(* CODESYS project sensata_device_comm.library
   Company: Sensata Technologies
   Version: 0.0.1
   DocFormat: reStructuredText
   Placeholder: Sensata_Device_Comm
   Title: Sensata_Device_Comm

Project tree, tasks and I/O mapping:
  libraries: Sensata_Common, * (Sensata Technologies); Sensata_Utilities, * (Sensata Technologies); Tc2_Standard, * (Beckhoff Automation GmbH); Tc2_System, * (Beckhoff Automation GmbH); Tc2_Utilities, * (Beckhoff Automation GmbH); Tc3_Module, * (Beckhoff Automation GmbH)
  Abstract/
    function block FB_Device_Comm [ST]: M_init, M_LoadDevice, M_PowerDown, M_PowerUp, M_ReadDeviceOP, M_ReadSerialNumber, M_RunCommand, M_RunImpMethods, M_SetCurrentDevice
  Concrete/
    data type E_COHAP_Error
    function block FB_COHAP [ST]: M_init, M_LoadDevice, M_PowerDown, M_PowerUp, M_ReadDeviceOP, M_ReadSerialNumber, M_SetCurrentDevice, A_CommandRecovery, M_ParseValue, M_RouterHelper, M_RunCommand, M_RunImpMethods
  Interfaces/
    interface I_DeviceCommunicable: M_init, M_LoadDevice, M_PowerDown, M_PowerUp, M_ReadDeviceOP, M_ReadSerialNumber
  Project Information/
    function F_GetCompany [ST]
    function F_GetTitle [ST]
    function F_GetVersion [ST]
  Version/
    global variables Global_Version
  data type E_DataType
  data type ReturnParamKVP
  data type ST_CohapParam
  data type T_CohapParameterList
*)

// Concrete/E_COHAP_Error
{attribute 'qualified_only'}
{attribute 'strict'}
TYPE E_COHAP_Error :
(
	None := 0,
	
	CommandRouterError			:= 0100, // Error on the command router FB
	CommandFault 				:= 0101, // Command failed to execute
	
	FailedToLoadDevice 			:= 0200, // Unable Load new device information
	
	FailedToReadSerialNum		:=0300,// Read Serial num Fail
	FailedToReadDeviceOP		:=0301,// Read Device Op Fail
	FailedToPowerUp 			:= 0400, // Unable Load new device information
	FailedToPowerDown 			:= 0401, // Unable Load new device information
	
	FailedToRunImpMethods		:= 0500, //Unable to succesfully execute the runimpMethods function on DeviceComm CohapDevice.cs class
	FailedToExecuteRunCommand   := 0501  //Unable to execute the execute the RunCommand function on DeviceComm CohapDevice.cs class for the functionality we require
	
)UDINT;
END_TYPE

// E_DataType
TYPE E_DataType : (
    DT_INT,
    DT_REAL,
    DT_BOOL,
    DT_STRING,
    DT_DINT,
    DT_UDINT,
	DT_DATETIME,
	DT_DOUBLE,
	DT_INT64,
	DT_UINT,
	DT_ULINT //This is 64 bit equivalent
    // Add more as needed
);
END_TYPE

// ReturnParamKVP
TYPE ReturnParamKVP :
STRUCT
	VarName: STRING; // Key - Variable name
	DataType: E_DataType; // Value - Data type
END_STRUCT
END_TYPE

// ST_CohapParam
TYPE ST_CohapParam :
STRUCT
	strKey : T_MaxString;
	strValue : T_MaxString;//T_ApiParamValue;//T_MaxString;
END_STRUCT
END_TYPE

// T_CohapParameterList
TYPE T_CohapParameterList : ARRAY[0..9] OF ST_CohapParam; END_TYPE

// Version/Global_Version
{attribute 'TcGenerated'}
{attribute 'no-analysis'}
{attribute 'linkalways'}
// This function has been automatically generated from the project information.
VAR_GLOBAL CONSTANT
	{attribute 'const_non_replaced'}
	stLibVersion_Sensata_ASIC_Comm : ST_LibVersion := (iMajor := 0, iMinor := 0, iBuild := 1, iRevision := 0, nFlags := 0, sVersion := '0.0.1');
END_VAR

// Abstract/FB_Device_Comm
FUNCTION_BLOCK ABSTRACT FB_Device_Comm EXTENDS FB_Device IMPLEMENTS  I_DeviceCommunicable

VAR_INPUT
END_VAR
VAR_OUTPUT
END_VAR
VAR
END_VAR

{warning 'add method implementation '}
METHOD M_init : BOOL
VAR_INPUT
	(*channel*)
	udintChannel	: UDINT;
END_VAR
END_METHOD


METHOD M_LoadDevice : BOOL
VAR_INPUT
    strDevName: STRING ;//Device Name
END_VAR
END_METHOD


METHOD M_PowerDown : BOOL
VAR_INPUT
	str_devID: STRING;	
	Channel_Num:UDINT;
END_VAR
END_METHOD


METHOD M_PowerUp : BOOL
VAR_INPUT
	str_devID: STRING;	
	Channel_Num:UDINT;
	lrVsupply :LREAL;
	udintSalveadd: UDINT;

END_VAR
VAR_OUTPUT
	voltage: LREAL;	
	current:LREAL;
END_VAR
END_METHOD


METHOD M_ReadDeviceOP : BOOL
VAR_INPUT
	(* String representing Device ID *)
	str_deviceID: STRING;
	Channel_Num: UDINT;
END_VAR

VAR_OUTPUT
	(*  representing device op *)
	udint_MeasuredTemp: UDINT;
	udint_MeasuredPressure: UDINT;
END_VAR
M_ReadDeviceOP := TRUE;
THIS^.M_LogWarning('M_ReadDeviceOP not implemented!');
END_METHOD


METHOD M_ReadSerialNumber : BOOL
VAR_INPUT
	(* String representing Device ID *)
	str_deviceID: STRING;
	Channel_Num: UDINT;
END_VAR

VAR_OUTPUT
	(* udint representing read serial num from the device*)
	udintSerialNum: UDINT;
END_VAR
M_ReadSerialNumber := TRUE;
THIS^.M_LogWarning('M_ReadSerialNumber not implemented!');
END_METHOD

METHOD PUBLIC ABSTRACT M_RunCommand : BOOL
VAR_INPUT
	 strMethod :STRING;
	 aInputParam :T_CohapParameterList;//T_ApiParameterList//T_CohapParameterList
	 aExpectedOutputParamsList : ARRAY[0..9] OF ReturnParamKVP; // Adjust size as necessary;
END_VAR
VAR_OUTPUT
	 aoutputParam :T_CohapParameterList;//T_ApiParameterList//T_CohapParameterList
END_VAR
END_METHOD

METHOD PUBLIC ABSTRACT M_RunImpMethods : BOOL
VAR_INPUT
END_VAR
END_METHOD

METHOD PUBLIC ABSTRACT M_SetCurrentDevice : BOOL
VAR_INPUT
    strDevName: STRING ;//Device Name
END_VAR
END_METHOD

END_FUNCTION_BLOCK

// Interfaces/I_DeviceCommunicable
INTERFACE I_DeviceCommunicable

METHOD M_init : BOOL
VAR_INPUT
    udintChannel: UDINT ;//channel
END_VAR
END_METHOD

METHOD M_LoadDevice : BOOL
VAR_INPUT
    strDevName: STRING ;//Device Name
END_VAR
END_METHOD

METHOD M_PowerDown : BOOL
VAR_INPUT
	str_devID: STRING;	
	Channel_Num:UDINT;
END_VAR
END_METHOD

METHOD M_PowerUp : BOOL

VAR_INPUT
	str_devID: STRING;	
	Channel_Num:UDINT;
	lrVsupply :LREAL;
	udintSalveadd: UDINT;
	
END_VAR
VAR_OUTPUT
	voltage: LREAL;	
	current:LREAL;
END_VAR
END_METHOD

METHOD M_ReadDeviceOP : BOOL
VAR_INPUT
	(* String representing Device ID *)
	str_deviceID: STRING;
	Channel_Num: UDINT;
END_VAR

VAR_OUTPUT
	(*  representing device op *)
	udint_MeasuredTemp: UDINT;
	udint_MeasuredPressure: UDINT;
END_VAR
END_METHOD

METHOD M_ReadSerialNumber : BOOL
VAR_INPUT
	(* String representing Device ID *)
	str_deviceID: STRING;
	Channel_Num: UDINT;
END_VAR

VAR_OUTPUT
	(* udint representing read serial num from the device*)
	udintSerialNum: UDINT;
END_VAR
END_METHOD

END_INTERFACE

// Concrete/FB_COHAP
FUNCTION_BLOCK FB_COHAP EXTENDS FB_Device_Comm IMPLEMENTS  I_DeviceCommunicable

VAR_INPUT
	(* Reference to an FB_CommandRouter function block to send commands
		to a command router in the API. *)
	fbApi : REFERENCE TO FB_CommandRouter;
END_VAR
VAR_OUTPUT
END_VAR
VAR
	
// Connectable
	bApiConnected: BOOL; (* TRUE if the API is connected. *)
	bConnected: BOOL; (* TRUE if the hipot is connected. *)
	bConnecting: BOOL; (* TRUE while the connect command is running. *)
	bDisconnecting: BOOL; (* TRUE while the disconnect command is running. *)
	
	enumProgramState: E_PROGRAMSTATE; // Value of P_enumProgramState
	bRouterBusy: BOOL; // TRUE while M_RouterHelper is being used by a method
	bResetBusy: BOOL; // Value of P_bResetBusy
	
	
	intInitStep: INT;
	intLoadDeviceStep: INT;
	intPowerUpStep: INT;
	intPowerDownStep: INT;
	intReadDeviceOPStep: INT;
	intReadDeviceSNStep: INT;
	intRouterHelperStep: INT;
	intMSetCurrentDeviceStep : INT;
	intMRunCommandStep : INT;
	intMRunImpMethodsStep : INT;
	
	
	bLoadDeviceBusy: BOOL;
	bInitBusy: BOOL;
	bPowerUpBusy: BOOL;
	bPowerDownBusy: BOOL;
	bReadDeviceOPBusy:BOOL;
	bReadDeviceSerialNumberBusy:BOOL;
	bRouterHelperBusy: BOOL;
	bSetCurrentDeviceBusy : BOOL;
	bMRunCommandBusy : BOOL;
	bRunImpMethodsBusy : BOOL;
	
END_VAR


A_CommandRecovery();

METHOD M_init : BOOL
VAR_INPUT
    udintChannel: UDINT ;//channel
END_VAR

VAR CONSTANT
	_strCOMMAND_NAME : T_MaxString	:= 'init'; // Name of the API method
	_timeCOMMAND_TIMEOUT : TIME		:= T#5S; // Max time to receive API response
	_strSTART_MSG : T_MaxString		:= 'initializing DUT '; // Prints when method starts
	_strEND_MSG : T_MaxString		:= 'DUT structure initialized'; // Prints when method finishes
	_udintERROR_ID : UDINT			:= E_COHAP_Error.FailedToLoadDevice; // Error ID to set if command fails
	_strERROR_MSG : T_MaxString		:= 'Failed to initialize!'; // Error message to set if command fails
END_VAR
VAR_INST
	_inst_arrParams: T_ApiParameterList; // Parameters array
	_inst_arrOutputs: T_ApiParameterList; // Outputs array
	_inst_strRet: T_ApiParamValue; // Return string from the router
	_inst_intStep: INT; // Current method step
	_inst_fbParams: FB_ApiParamBuilder; // Parameter builder FB
END_VAR
VAR
	_bComplete: BOOL; // True if the routing finishes
	_intRet: INT; // Return string converted to an integer
	_bResult : BOOL; // Output of the method
END_VAR
_inst_intStep:=intInitStep;
bInitBusy:=TRUE;

_bResult:=FALSE;
CASE _inst_intStep OF
	0: // Wait for no error and router not busy
		IF NOT THIS^.P_bError AND NOT bRouterBusy THEN
			bRouterBusy := TRUE;
			_inst_intStep := _inst_intStep + 10;
		END_IF
		
	10: // Initialize parameters
		THIS^.M_LogMessage(_strSTART_MSG);
		_inst_fbParams.M_ClearParameters();
		// ADD ANY PARAMETERS HERE
		_inst_fbParams.M_AddParameter('channel', udintChannel);
		
		_inst_fbParams.M_OutputToParameterList(_inst_arrParams);
		_inst_intStep := _inst_intStep + 10;
		
	20: // Route the command
		_bComplete := M_RouterHelper(
			_in_strMethodName := _strCOMMAND_NAME, 
			_in_timeTimeout := _timeCOMMAND_TIMEOUT,
			_inout_arrParams := _inst_arrParams,
			_inout_arrOutputs := _inst_arrOutputs,
			_out_strReturnValue=>_inst_strRet);
		
		// If route completed, move to next step
		IF _bComplete THEN
			_inst_intStep := _inst_intStep + 10;
			bRouterBusy := FALSE;
		ELSIF THIS^.P_bError THEN
			_inst_intStep := 0;
			bRouterBusy := FALSE;
		END_IF
		
	30: // Parse results
		_intRet := STRING_TO_INT(_inst_strRet);
		IF _intRet > 0 THEN
			_bResult := TRUE;
			THIS^.M_LogMessage(_strEND_MSG);
			// DO ANY PARSING HERE
			_inst_fbParams.M_LoadFromParameterList(_inst_arrOutputs);
		
		// Set error if command failed
	
		ELSE
			THIS^.M_SetError(_udintERROR_ID, _strERROR_MSG);
		END_IF
		
		// Go back to start
		_inst_intStep := 0;
END_CASE
M_init := _bResult;
intInitStep:=_inst_intStep;
END_METHOD

METHOD M_LoadDevice : BOOL
VAR_INPUT
    strDevName: STRING ;//Device Name
END_VAR

VAR CONSTANT
	_strCOMMAND_NAME : T_MaxString	:= 'LoadDevice'; // Name of the API method
	_timeCOMMAND_TIMEOUT : TIME		:= T#5S; // Max time to receive API response
	_strSTART_MSG : T_MaxString		:= 'Load a new device to test'; // Prints when method starts
	_strEND_MSG : T_MaxString		:= 'Device details loaded'; // Prints when method finishes
	_udintERROR_ID : UDINT			:= E_COHAP_Error.FailedToLoadDevice; // Error ID to set if command fails
	_strERROR_MSG : T_MaxString		:= 'Failed to connect!'; // Error message to set if command fails
END_VAR
VAR_INST
	_inst_arrParams: T_ApiParameterList; // Parameters array
	_inst_arrOutputs: T_ApiParameterList; // Outputs array
	_inst_strRet: T_ApiParamValue; // Return string from the router
	_inst_intStep: INT; // Current method step
	_inst_fbParams: FB_ApiParamBuilder; // Parameter builder FB
END_VAR
VAR
	_bComplete: BOOL; // True if the routing finishes
	_intRet: INT; // Return string converted to an integer
	_bResult : BOOL; // Output of the method
END_VAR
_inst_intStep:=intLoadDeviceStep;
bLoadDeviceBusy:=TRUE;

_bResult := FALSE;
CASE _inst_intStep OF
	0: // Wait for no error and router not busy
		IF NOT THIS^.P_bError AND NOT bRouterBusy THEN
			bRouterBusy := TRUE;
			_inst_intStep := _inst_intStep + 10;
		END_IF
		
	10: // Initialize parameters
		THIS^.M_LogMessage(_strSTART_MSG);
		_inst_fbParams.M_ClearParameters();
		// ADD ANY PARAMETERS HERE
		_inst_fbParams.M_AddParameter('devID', strDevName);
		
		_inst_fbParams.M_OutputToParameterList(_inst_arrParams);
		_inst_intStep := _inst_intStep + 10;
		
	20: // Route the command
		_bComplete := M_RouterHelper(
			_in_strMethodName := _strCOMMAND_NAME, 
			_in_timeTimeout := _timeCOMMAND_TIMEOUT,
			_inout_arrParams := _inst_arrParams,
			_inout_arrOutputs := _inst_arrOutputs,
			_out_strReturnValue=>_inst_strRet);
		
		// If route completed, move to next step
		IF _bComplete THEN
			_inst_intStep := _inst_intStep + 10;
			bRouterBusy := FALSE;
		ELSIF THIS^.P_bError THEN
			_inst_intStep := 0;
			bRouterBusy := FALSE;
		END_IF
		
	30: // Parse results
		_intRet := STRING_TO_INT(_inst_strRet);
		IF _intRet > 0 THEN
			_bResult := TRUE;
			THIS^.M_LogMessage(_strEND_MSG);
			// DO ANY PARSING HERE
			_inst_fbParams.M_LoadFromParameterList(_inst_arrOutputs);
		
		// Set error if command failed
	
		ELSE
			THIS^.M_SetError(_udintERROR_ID, _strERROR_MSG);
		END_IF
		
		// Go back to start
		_inst_intStep := 0;
END_CASE
M_LoadDevice := _bResult;
intLoadDeviceStep:=_inst_intStep;
END_METHOD


METHOD M_PowerDown : BOOL
VAR_INPUT
	str_devID: STRING;	
	Channel_Num:UDINT;

END_VAR
VAR CONSTANT
	_strCOMMAND_NAME : T_MaxString	:= 'Powerdown'; // Name of the API method
	_timeCOMMAND_TIMEOUT : TIME		:= T#5S; // Max time to receive API response
	_strSTART_MSG : T_MaxString		:= 'Powering Down device'; // Prints when method starts
	_strEND_MSG : T_MaxString		:= 'Device Powered Down'; // Prints when method finishes
	_udintERROR_ID : UDINT			:= E_COHAP_Error.FailedToPowerDown; // Error ID to set if command fails
	_strERROR_MSG : T_MaxString		:= 'Failed to Power Down!'; // Error message to set if command fails
END_VAR
VAR_INST
	_inst_arrParams: T_ApiParameterList; // Parameters array
	_inst_arrOutputs: T_ApiParameterList; // Outputs array
	_inst_strRet: T_ApiParamValue; // Return string from the router
	_inst_intStep: INT; // Current method step
	_inst_fbParams: FB_ApiParamBuilder; // Parameter builder FB
END_VAR
VAR
	_bComplete: BOOL; // True if the routing finishes
	_intRet: INT; // Return string converted to an integer
	_bResult : BOOL; // Output of the method
END_VAR
_inst_intStep := intPowerDownStep;
bPowerDownBusy := TRUE;

_bResult := FALSE;
CASE _inst_intStep OF
	0: // Wait for no error and router not busy
		IF NOT THIS^.P_bError AND NOT bRouterBusy THEN
			bRouterBusy := TRUE;
			_inst_intStep := _inst_intStep + 10;
		END_IF
		
	10: // Initialize parameters
		THIS^.M_LogMessage(_strSTART_MSG);
		_inst_fbParams.M_ClearParameters();
		// ADD ANY PARAMETERS HERE
		
		_inst_fbParams.M_AddParameter('devID', str_devID);
		_inst_fbParams.M_AddParameter('channel', Channel_Num);
		_inst_fbParams.M_OutputToParameterList(_inst_arrParams);
		_inst_intStep := _inst_intStep + 10;
		
	20: // Route the command
		_bComplete := M_RouterHelper(
			_in_strMethodName := _strCOMMAND_NAME, 
			_in_timeTimeout := _timeCOMMAND_TIMEOUT,
			_inout_arrParams := _inst_arrParams,
			_inout_arrOutputs := _inst_arrOutputs,
			_out_strReturnValue=>_inst_strRet);
		
		// If route completed, move to next step
		IF _bComplete THEN
			_inst_intStep := _inst_intStep + 10;
			bRouterBusy := FALSE;
		ELSIF THIS^.P_bError THEN
			_inst_intStep := 0;
			bRouterBusy := FALSE;
		END_IF
		
	30: // Parse results
		_intRet := STRING_TO_INT(_inst_strRet);
		IF _intRet > 0 THEN
			_bResult := TRUE;
			THIS^.M_LogMessage(_strEND_MSG);
			// DO ANY PARSING HERE
			_inst_fbParams.M_LoadFromParameterList(_inst_arrOutputs);
		
		// Set error if command failed
	
		ELSE
			THIS^.M_SetError(_udintERROR_ID, _strERROR_MSG);
		END_IF
		
		// Go back to start
		_inst_intStep := 0;
END_CASE
M_PowerDown := _bResult;
intPowerDownStep:=_inst_intStep;
END_METHOD

METHOD M_PowerUp : BOOL
VAR_INPUT
	str_devID: STRING;	
	Channel_Num:UDINT;
	lrVsupply :LREAL;
	udintSalveadd: UDINT;
END_VAR
VAR_OUTPUT
	voltage: LREAL;	
	current:LREAL;
END_VAR
VAR CONSTANT
	_strCOMMAND_NAME : T_MaxString	:= 'Powerup'; // Name of the API method
	_timeCOMMAND_TIMEOUT : TIME		:= T#5S; // Max time to receive API response
	_strSTART_MSG : T_MaxString		:= 'Powering Up device'; // Prints when method starts
	_strEND_MSG : T_MaxString		:= 'Device Powered Up'; // Prints when method finishes
	_udintERROR_ID : UDINT			:= E_COHAP_Error.FailedToPowerUp; // Error ID to set if command fails
	_strERROR_MSG : T_MaxString		:= 'Failed to Power Up!'; // Error message to set if command fails
END_VAR
VAR_INST
	_inst_arrParams: T_ApiParameterList; // Parameters array
	_inst_arrOutputs: T_ApiParameterList; // Outputs array
	_inst_strRet: T_ApiParamValue; // Return string from the router
	_inst_intStep: INT; // Current method step
	_inst_fbParams: FB_ApiParamBuilder; // Parameter builder FB
END_VAR
VAR
	_bComplete: BOOL; // True if the routing finishes
	_intRet: INT; // Return string converted to an integer
	_bResult : BOOL; // Output of the method
END_VAR
_inst_intStep := intPowerUpStep;
bPowerUpBusy := TRUE;

_bResult := FALSE;
CASE _inst_intStep OF
	0: // Wait for no error and router not busy
		IF NOT THIS^.P_bError AND NOT bRouterBusy THEN
			bRouterBusy := TRUE;
			_inst_intStep := _inst_intStep + 10;
		END_IF
		
	10: // Initialize parameters
		THIS^.M_LogMessage(_strSTART_MSG);
		_inst_fbParams.M_ClearParameters();
		// ADD ANY PARAMETERS HERE
		
		_inst_fbParams.M_AddParameter('devID', str_devID);
		_inst_fbParams.M_AddParameter('channel', Channel_Num);
		_inst_fbParams.M_AddParameter('VSupply', lrVsupply);
		_inst_fbParams.M_AddParameter('slaveadd', udintSalveadd);
		_inst_fbParams.M_OutputToParameterList(_inst_arrParams);
		_inst_intStep := _inst_intStep + 10;
		
	20: // Route the command
		_bComplete := M_RouterHelper(
			_in_strMethodName := _strCOMMAND_NAME, 
			_in_timeTimeout := _timeCOMMAND_TIMEOUT,
			_inout_arrParams := _inst_arrParams,
			_inout_arrOutputs := _inst_arrOutputs,
			_out_strReturnValue=>_inst_strRet);
		
		// If route completed, move to next step
		IF _bComplete THEN
			_inst_intStep := _inst_intStep + 10;
			bRouterBusy := FALSE;
		ELSIF THIS^.P_bError THEN
			_inst_intStep := 0;
			bRouterBusy := FALSE;
		END_IF
		
	30: // Parse results
		_intRet := STRING_TO_INT(_inst_strRet);
		IF _intRet > 0 THEN
			_bResult := TRUE;
			THIS^.M_LogMessage(_strEND_MSG);
			// DO ANY PARSING HERE
			_inst_fbParams.M_LoadFromParameterList(_inst_arrOutputs);
			voltage := _inst_fbParams.M_ParseDouble(_inst_fbParams.M_GetParameter('Respvoltage'));
			current := _inst_fbParams.M_ParseDouble(_inst_fbParams.M_GetParameter('Respcurrent'));
		// Set error if command failed
	
		ELSE
			THIS^.M_SetError(_udintERROR_ID, _strERROR_MSG);
		END_IF
		
		// Go back to start
		_inst_intStep := 0;
END_CASE
M_PowerUp := _bResult;
intPowerUpStep:=_inst_intStep;
END_METHOD


(* This method takes deviceID as input as passes it to the COHAP API library to get the Device OP *)
METHOD M_ReadDeviceOP : BOOL
VAR_INPUT
	(* String representing Device ID *)
	str_deviceID: STRING;
	Channel_Num: UDINT;
END_VAR

VAR_OUTPUT
	(*  representing device op *)
	udint_MeasuredTemp: UDINT;
	udint_MeasuredPressure: UDINT;
END_VAR
VAR CONSTANT
	_strCOMMAND_NAME : T_MaxString	:= 'ReadDeviceOutput'; // Name of the API method
	_timeCOMMAND_TIMEOUT : TIME		:= T#7S; // Max time to receive API response
	_strSTART_MSG : T_MaxString		:= 'Reading Device output'; // Prints when method starts
	_strEND_MSG : T_MaxString		:= 'Completed device OP read'; // Prints when method finishes
	_udintERROR_ID : UDINT			:= E_COHAP_Error.FailedToReadDeviceOP; // Error ID to set if command fails
	_strERROR_MSG : T_MaxString		:= 'Failed to read Device output!'; // Error message to set if command fails
END_VAR
VAR_INST
	_inst_arrParams: T_ApiParameterList; // Parameters array
	_inst_arrOutputs: T_ApiParameterList; // Outputs array
	_inst_strRet: T_ApiParamValue; // Return string from the router
	_inst_intStep: INT; // Current method step
	_inst_fbParams: FB_ApiParamBuilder; // Parameter builder FB
END_VAR
VAR
	_bComplete: BOOL; // True if the routing finishes
	_intRet: INT; // Return string converted to an integer
	_bResult : BOOL; // Output of the method
END_VAR
_inst_intStep := intReadDeviceOPStep;
bReadDeviceOPBusy := TRUE;

_bResult := FALSE;
CASE _inst_intStep OF
	0: // Wait for no error and router not busy
		IF NOT THIS^.P_bError AND NOT bRouterBusy THEN
			bRouterBusy := TRUE;
			_inst_intStep := _inst_intStep + 10;
		END_IF
		
	10: // Initialize parameters
		THIS^.M_LogMessage(_strSTART_MSG);
		_inst_fbParams.M_ClearParameters();
		// ADD ANY PARAMETERS HERE
		_inst_fbParams.M_AddParameter('DeviceID', str_deviceID);
		_inst_fbParams.M_AddParameter('channel', Channel_Num);
		_inst_fbParams.M_OutputToParameterList(_inst_arrParams);
		_inst_intStep := _inst_intStep + 10;
		
	20: // Route the command
		_bComplete := M_RouterHelper(
			_in_strMethodName := _strCOMMAND_NAME, 
			_in_timeTimeout := _timeCOMMAND_TIMEOUT,
			_inout_arrParams := _inst_arrParams,
			_inout_arrOutputs := _inst_arrOutputs,
			_out_strReturnValue=>_inst_strRet);
		
		// If route completed, move to next step
		IF _bComplete THEN
			_inst_intStep := _inst_intStep + 10;
			bRouterBusy := FALSE;
		ELSIF THIS^.P_bError THEN
			_inst_intStep := 0;
			bRouterBusy := FALSE;
		END_IF
		
	30: // Parse results
		_intRet := STRING_TO_INT(_inst_strRet);
		IF _intRet > 0 THEN
			_bResult := TRUE;
			THIS^.M_LogMessage(_strEND_MSG);
			// DO ANY PARSING HERE
			_inst_fbParams.M_LoadFromParameterList(_inst_arrOutputs);
			udint_MeasuredTemp := _inst_fbParams.M_ParseUint(_inst_fbParams.M_GetParameter('OutputTemp'));
			udint_MeasuredPressure := _inst_fbParams.M_ParseUint(_inst_fbParams.M_GetParameter('OutputPress'));		
		// Set error if command failed
	
		ELSE
			THIS^.M_SetError(_udintERROR_ID, _strERROR_MSG);
		END_IF
		
		// Go back to start
		_inst_intStep := 0;
END_CASE
M_ReadDeviceOP := _bResult;
intReadDeviceOPStep:=_inst_intStep;
END_METHOD




(* This method takes deviceID as input as passes it to the COHAP API library to get the serial number *)
METHOD M_ReadSerialNumber : BOOL
VAR_INPUT
	(* String representing Device ID *)
	str_deviceID: STRING;
	Channel_Num: UDINT;

END_VAR

VAR_OUTPUT
	(* udint representing read serial num from the device*)
	udintSerialNum: UDINT;
END_VAR
VAR CONSTANT
	_strCOMMAND_NAME : T_MaxString	:= 'ReadSerialNumber'; // Name of the API method
	_timeCOMMAND_TIMEOUT : TIME		:= T#7S; // Max time to receive API response
	_strSTART_MSG : T_MaxString		:= 'Reading Device Serialnumber'; // Prints when method starts
	_strEND_MSG : T_MaxString		:= 'Completed Serial Num read'; // Prints when method finishes
	_udintERROR_ID : UDINT			:= E_COHAP_Error.FailedToReadSerialNum; // Error ID to set if command fails
	_strERROR_MSG : T_MaxString		:= 'Failed to read serial number!'; // Error message to set if command fails
END_VAR
VAR_INST
	_inst_arrParams: T_ApiParameterList; // Parameters array
	_inst_arrOutputs: T_ApiParameterList; // Outputs array
	_inst_strRet: T_ApiParamValue; // Return string from the router
	_inst_intStep: INT; // Current method step
	_inst_fbParams: FB_ApiParamBuilder; // Parameter builder FB
END_VAR
VAR
	_bComplete: BOOL; // True if the routing finishes
	_intRet: INT; // Return string converted to an integer
	_bResult : BOOL; // Output of the method
END_VAR
_inst_intStep := intReadDeviceSNStep;
bReadDeviceSerialNumberBusy := TRUE;

_bResult := FALSE;
CASE _inst_intStep OF
	0: // Wait for no error and router not busy
		IF NOT THIS^.P_bError AND NOT bRouterBusy THEN
			bRouterBusy := TRUE;
			_inst_intStep := _inst_intStep + 10;
		END_IF
		
	10: // Initialize parameters
		THIS^.M_LogMessage(_strSTART_MSG);
		_inst_fbParams.M_ClearParameters();
		// ADD ANY PARAMETERS HERE
		_inst_fbParams.M_AddParameter('DeviceID', str_deviceID);
		_inst_fbParams.M_AddParameter('channel', Channel_Num);
		_inst_fbParams.M_OutputToParameterList(_inst_arrParams);
		_inst_intStep := _inst_intStep + 10;
		
	20: // Route the command
		_bComplete := M_RouterHelper(
			_in_strMethodName := _strCOMMAND_NAME, 
			_in_timeTimeout := _timeCOMMAND_TIMEOUT,
			_inout_arrParams := _inst_arrParams,
			_inout_arrOutputs := _inst_arrOutputs,
			_out_strReturnValue=>_inst_strRet);
		
		// If route completed, move to next step
		IF _bComplete THEN
			_inst_intStep := _inst_intStep + 10;
			bRouterBusy := FALSE;
		ELSIF THIS^.P_bError THEN
			_inst_intStep := 0;
			bRouterBusy := FALSE;
		END_IF
		
	30: // Parse results
		_intRet := STRING_TO_INT(_inst_strRet);
		IF _intRet > 0 THEN
			_bResult := TRUE;
			THIS^.M_LogMessage(_strEND_MSG);
			// DO ANY PARSING HERE
			_inst_fbParams.M_LoadFromParameterList(_inst_arrOutputs);
			udintSerialNum := _inst_fbParams.M_ParseUint(_inst_fbParams.M_GetParameter('serialNumber'));
					
		// Set error if command failed
	
		ELSE
			THIS^.M_SetError(_udintERROR_ID, _strERROR_MSG);
		END_IF
		
		// Go back to start
		_inst_intStep := 0;
END_CASE
M_ReadSerialNumber := _bResult;
intReadDeviceSNStep:=_inst_intStep;
END_METHOD

METHOD M_SetCurrentDevice : BOOL
VAR_INPUT
    strDevName: STRING ;//Device Name
END_VAR

VAR CONSTANT
	_strCOMMAND_NAME : T_MaxString	:= 'SetCurrentDevice'; // Name of the API method
	_timeCOMMAND_TIMEOUT : TIME		:= T#30S; // Max time to receive API response
	_strSTART_MSG : T_MaxString		:= 'Load a new device to test'; // Prints when method starts
	_strEND_MSG : T_MaxString		:= 'Device details loaded'; // Prints when method finishes
	_udintERROR_ID : UDINT			:= E_COHAP_Error.FailedToLoadDevice; // Error ID to set if command fails
	_strERROR_MSG : T_MaxString		:= 'Failed to connect!'; // Error message to set if command fails
END_VAR
VAR_INST
	_inst_arrParams: T_ApiParameterList; // Parameters array
	_inst_arrOutputs: T_ApiParameterList; // Outputs array
	_inst_strRet: T_ApiParamValue; // Return string from the router
	_inst_intStep: INT; // Current method step
	_inst_fbParams: FB_ApiParamBuilder; // Parameter builder FB
END_VAR
VAR
	_bComplete: BOOL; // True if the routing finishes
	_intRet: INT; // Return string converted to an integer
	_bResult : BOOL; // Output of the method
END_VAR
_inst_intStep := intMSetCurrentDeviceStep;
bSetCurrentDeviceBusy := TRUE;

_bResult := FALSE;
CASE _inst_intStep OF
	0: // Wait for no error and router not busy
		IF NOT THIS^.P_bError AND NOT bRouterBusy THEN
			bRouterBusy := TRUE;
			_inst_intStep := _inst_intStep + 10;
		END_IF
		
	10: // Initialize parameters
		THIS^.M_LogMessage(_strSTART_MSG);
		_inst_fbParams.M_ClearParameters();
		// ADD ANY PARAMETERS HERE
		_inst_fbParams.M_AddParameter('DeviceName', strDevName);
		
		_inst_fbParams.M_OutputToParameterList(_inst_arrParams);
		_inst_intStep := _inst_intStep + 10;
		
	20: // Route the command
		_bComplete := M_RouterHelper(
			_in_strMethodName := _strCOMMAND_NAME, 
			_in_timeTimeout := _timeCOMMAND_TIMEOUT,
			_inout_arrParams := _inst_arrParams,
			_inout_arrOutputs := _inst_arrOutputs,
			_out_strReturnValue=>_inst_strRet);
		
		// If route completed, move to next step
		IF _bComplete THEN
			_inst_intStep := _inst_intStep + 10;
			bRouterBusy := FALSE;
		ELSIF THIS^.P_bError THEN
			_inst_intStep := 0;
			bRouterBusy := FALSE;
		END_IF
		
	30: // Parse results
		_intRet := STRING_TO_INT(_inst_strRet);
		IF _intRet > 0 THEN
			_bResult := TRUE;
			THIS^.M_LogMessage(_strEND_MSG);
			// DO ANY PARSING HERE
			_inst_fbParams.M_LoadFromParameterList(_inst_arrOutputs);
			
					
		// Set error if command failed
	
		ELSE
			THIS^.M_SetError(_udintERROR_ID, _strERROR_MSG);
		END_IF
		
		// Go back to start
		_inst_intStep := 0;
END_CASE
M_SetCurrentDevice := _bResult;
intMSetCurrentDeviceStep := _inst_intStep;
END_METHOD

ACTION A_CommandRecovery:
IF NOT bInitBusy AND intInitStep > 0 THEN
	intInitStep := 0;
	bRouterBusy := FALSE;
	THIS^.M_LogWarning('Init ended prematurely!');
END_IF
bInitBusy := FALSE;

IF NOT bLoadDeviceBusy AND intLoadDeviceStep > 0 THEN
	intLoadDeviceStep := 0;
	bRouterBusy := FALSE;
	THIS^.M_LogWarning('LoadDevice ended prematurely!');
END_IF
bLoadDeviceBusy := FALSE;

IF NOT bPowerDownBusy AND intPowerDownStep > 0 THEN
	intPowerDownStep := 0;
	bRouterBusy := FALSE;
	THIS^.M_LogWarning('PowerDown ended prematurely!');
END_IF
bPowerDownBusy := FALSE;

IF NOT bPowerUpBusy AND intPowerUpStep > 0 THEN
	intPowerUpStep := 0;
	bRouterBusy := FALSE;
	THIS^.M_LogWarning(' Power up ended prematurely!');
END_IF
bPowerUpBusy := FALSE;

IF NOT bReadDeviceOPBusy AND intReadDeviceOPStep > 0 THEN
	intReadDeviceOPStep := 0;
	bRouterBusy := FALSE;
	THIS^.M_LogWarning('Read Device  OP ended prematurely!');
END_IF
bReadDeviceOPBusy := FALSE;

IF NOT bReadDeviceSerialNumberBusy AND intReadDeviceSNStep > 0 THEN
	intReadDeviceSNStep := 0;
	bRouterBusy := FALSE;
	THIS^.M_LogWarning('Read Serial Number ended prematurely!');
END_IF
bReadDeviceSerialNumberBusy := FALSE;

IF NOT bSetCurrentDeviceBusy AND intMSetCurrentDeviceStep > 0 THEN
	intMSetCurrentDeviceStep := 0;
	bRouterBusy := FALSE;
	THIS^.M_LogWarning('Set Current Device ended prematurely');
END_IF
bSetCurrentDeviceBusy := FALSE;

IF NOT bRunImpMethodsBusy AND intMRunImpMethodsStep > 0 THEN
	intMRunImpMethodsStep := 0;
	bRouterBusy := FALSE;
	THIS^.M_LogWarning('Run Imp Methods ended prematurely');
END_IF
bRunImpMethodsBusy := FALSE;

IF NOT bMRunCommandBusy AND intMRunCommandStep > 0 THEN
	intMRunCommandStep := 0;
	bRouterBusy := FALSE;
	THIS^.M_LogWarning('M_RunCommand ended prematurely!');
END_IF
bMRunCommandBusy := FALSE;

IF NOT bRouterHelperBusy AND intRouterHelperStep > 0 THEN
	intRouterHelperStep := 0;
	THIS^.M_LogWarning('Router helper ended prematurely!');
END_IF
bRouterHelperBusy := FALSE;
END_ACTION

METHOD M_ParseValue : BOOL
VAR_INPUT
    DataType : E_DataType; // The data type to which the value needs to be converted
    ValueStr : STRING;    // The value as a string
END_VAR
VAR_OUTPUT
    BoolValue    : BOOL;
    DateTimeValue: DT;    // Assuming DT is the datatype for DateTime
    DoubleValue  : REAL;
//    IntValue     : INT;
	DintValue 	 : DINT;
    Int64Value   : LINT;  // Assuming LINT is the datatype for 64-bit integer
    StringValue  : STRING;
//    UintValue    : UINT;
	UDINTValue   : UDINT;
    Uint64Value  : ULINT; // Assuming ULINT is the datatype for unsigned 64-bit integer
END_VAR
VAR
    ApiParamBuilder : FB_ApiParamBuilder;
    bResult         : BOOL := FALSE; // To store the success status of parsing
END_VAR
//CASE DataType OF
//    DT_BOOL:
//        BoolValue := ApiParamBuilder.M_ParseBool(ValueStr);
//    DT_DATETIME:
//        DateTimeValue := ApiParamBuilder.M_ParseDateTime(ValueStr);
        
//    DT_DOUBLE:
//        DoubleValue := ApiParamBuilder.M_ParseDouble(ValueStr);
        
//    DT_INT:
//        DIntValue := ApiParamBuilder.M_ParseInt(ValueStr);
        
//    DT_INT64:
//        Int64Value := ApiParamBuilder.M_ParseInt64(ValueStr);
        
//    DT_STRING:
//        StringValue := ApiParamBuilder.M_ParseString(ValueStr);
        
//    DT_UINT:
//        UDintValue := ApiParamBuilder.M_ParseUint(ValueStr);
        
//    DT_UINT64:
//        Uint64Value := ApiParamBuilder.M_ParseUint64(ValueStr);
        
//    ELSE
//        bResult := FALSE; // In case of an unrecognized data type
//END_CASE
END_METHOD

(*
Sends the given method to the API and receives and partially parses the result.
*)
METHOD PRIVATE M_RouterHelper : BOOL
VAR_INPUT
	(* Name of the method to call. *)
	_in_strMethodName : T_MaxString;
	(* Maximum time to wait for method response. *)
	_in_timeTimeout : TIME;
END_VAR
VAR_IN_OUT
	(* The array of parameters to send to the API. *)
	_inout_arrParams : T_ApiParameterList;
	(* The array that gets populated with any method output data. *)
	_inout_arrOutputs : T_ApiParameterList;
END_VAR
VAR_OUTPUT
	(* JSON string of the method return value. *)
	_out_strReturnValue: T_ApiParamValue;
END_VAR
VAR_INST
	(* Current step. *)
	_inst_intStep: INT;
	(* True if the method executed. *)
	_inst_bExec: BOOL;
	(* Return string of the method. *)
	_inst_strRet: T_ApiParamValue;
END_VAR
VAR
	(* True once the command routing finishes. *)
	_bComplete: BOOL;
	(* True once the API connects. *)
	_bApiConnect: BOOL;
END_VAR
_inst_intStep := intRouterHelperStep;
bRouterHelperBusy := TRUE;

CASE _inst_intStep OF
	0: // Start process only if there is no error on this FB
		IF NOT THIS^.P_bError THEN
			fbApi.M_ClearError();
			_inst_intStep := 10;
		END_IF
		
	10: // Check if command router connected
		IF NOT fbApi.P_bConnected THEN
			_inst_intStep := 20; // Go to API connect step
		ELSE
			_inst_intStep := 30; // Go to route command step
		END_IF
		
	20: // Connect the command router
		_bApiConnect := fbApi.M_Connect();
		IF _bApiConnect THEN
			_inst_intStep := _inst_intStep + 10; // Go to next step
		ELSIF fbApi.P_bError THEN
			THIS^.M_SetError(E_COHAP_Error.CommandRouterError, 'Error on command router function block while connecting!');
			_inst_intStep := 0; // Go back to start
		END_IF
		
	30:	// Route the command
		_bComplete := fbApi.M_RouteCommand(
			_in_strModuleId := in_strUniqueId,
			_in_strMethodName := _in_strMethodName,
			_in_timeTimeout := _in_timeTimeout,
			_inout_arrParameters := _inout_arrParams,
			_inout_arrOutputs := _inout_arrOutputs,
			_out_bCommandExecuted => _inst_bExec,
			_out_strReturnValue => _inst_strRet);
		IF _bComplete THEN
			_inst_intStep := _inst_intStep + 10; // Go to next step
		ELSIF fbApi.P_bError THEN
			THIS^.M_SetError(E_COHAP_Error.CommandRouterError, 'Error on command router function block while routing command!');
			_inst_intStep := 0; // Go back to start
		END_IF
		
	40: // Check result then go back to start
		IF NOT _inst_bExec THEN
			THIS^.M_SetError(E_COHAP_Error.CommandFault, 'Method in API failed to execute!');
		ELSE
			_out_strReturnValue := _inst_strRet;
			M_RouterHelper := TRUE;
		END_IF
		_inst_intStep := 0; // Go back to start
END_CASE

intRouterHelperStep := _inst_intStep;
END_METHOD

METHOD M_RunCommand : BOOL
VAR_INPUT
	 strMethod :STRING;
	 aInputParam :T_CohapParameterList;//T_ApiParameterList//T_CohapParameterList
	 aExpectedOutputParamsList : ARRAY[0..9] OF ReturnParamKVP; // Adjust size as necessary;
END_VAR
VAR_OUTPUT
	 aoutputParam :T_CohapParameterList;//T_ApiParameterList//T_CohapParameterList
END_VAR
VAR CONSTANT
	_strCOMMAND_NAME : T_MaxString	:= 'RunCommand'; // Name of the API method
	_timeCOMMAND_TIMEOUT : TIME		:= T#60S; // Max time to receive API response
	_strSTART_MSG : T_MaxString		:= 'Executing Run Command'; // Prints when method starts
	_strEND_MSG : T_MaxString		:= 'Completing the Execution of Run Command'; // Prints when method finishes
	_udintERROR_ID : UDINT			:= E_COHAP_Error.FailedToExecuteRunCommand; // Error ID to set if command fails
	_strERROR_MSG : T_MaxString		:= 'Failed to Execute the M_RunCommand function!'; // Error message to set if command fails
END_VAR
VAR_INST
	_inst_arrParams: T_ApiParameterList; // Parameters array
	_inst_arrOutputs: T_ApiParameterList; // Outputs array
	_inst_strRet: T_ApiParamValue; // Return string from the router
	_inst_intStep: INT; // Current method step
	_inst_fbParams: FB_ApiParamBuilder; // Parameter builder FB
	_inst_strlocal : STRING;
	 floatResponse : LREAL;
END_VAR
VAR
	_bComplete: BOOL; // True if the routing finishes
	_intRet: INT; // Return string converted to an integer
	_bResult : BOOL; // Output of the method
	stTempInpStruct: ST_AmsAddr;
	pStruct: PVOID;
	pStructOut:PVOID;
	_pStructPointer:PVOID;
	_pStructPointerAbs : PVOID;
	intIndex: INT;
	intValue : DINT;
	uintValue : UDINT;
	ulintValue : ULINT;
//	int64Value : uint
	boolresponse: BOOL;
END_VAR
_inst_intStep := intMRunCommandStep;
bMRunCommandBusy := TRUE;

_bResult := FALSE;
CASE _inst_intStep OF
	0: // Wait for no error and router not busy
		IF NOT THIS^.P_bError AND NOT bRouterBusy THEN
			bRouterBusy := TRUE;
			_inst_intStep := _inst_intStep + 10;
		END_IF
		
	10: // Initialize parameters
		THIS^.M_LogMessage(_strSTART_MSG);
		_inst_fbParams.M_ClearParameters();
		// ADD ANY PARAMETERS HERE
		
		_inst_fbParams.M_AddParameter('methodName', strMethod);
		pStruct := _inst_fbParams.M_AddEmptyStruct('input');
		FOR intIndex := 0 TO 9 DO
			IF aInputParam[intIndex].strKey <> '' THEN
				_inst_fbParams.M_AddStructMember(pStruct, aInputParam[intIndex].strKey, aInputParam[intIndex].strValue);
			END_IF
		END_FOR
		
		_inst_fbParams.M_OutputToParameterList(_inst_arrParams);
		_inst_intStep := _inst_intStep + 10;
		
	20: // Route the command
		_bComplete := M_RouterHelper(
			_in_strMethodName := _strCOMMAND_NAME, 
			_in_timeTimeout := _timeCOMMAND_TIMEOUT,
			_inout_arrParams := _inst_arrParams,
			_inout_arrOutputs := _inst_arrOutputs,
			_out_strReturnValue=>_inst_strRet);
		
		// If route completed, move to next step
		IF _bComplete THEN
			_inst_intStep := _inst_intStep + 10;
			bRouterBusy := FALSE;
		ELSIF THIS^.P_bError THEN
			_inst_intStep := 0;
			bRouterBusy := FALSE;
		END_IF
		
	30: // Parse results
		_intRet := STRING_TO_INT(_inst_strRet);
		IF _intRet > 0 THEN
			_bResult := TRUE;
			THIS^.M_LogMessage(_strEND_MSG);
			// DO ANY PARSING HERE
			_inst_fbParams.M_LoadFromParameterList(_inst_arrOutputs);
			_pStructPointer := _inst_fbParams.M_GetParameter('output');
			_pStructPointerAbs := _pStructPointer;
			FOR intIndex := 0 TO 9 DO
				IF aExpectedOutputParamsList[intIndex].VarName <> '' THEN
					aoutputParam[intIndex].strKey := aExpectedOutputParamsList[intIndex].VarName;
					IF aExpectedOutputParamsList[intIndex].DataType = E_DataType.DT_INT THEN
						intValue := _inst_fbParams.M_ParseInt(_inst_fbParams.M_GetStructMember(_pStructPointerAbs,aExpectedOutputParamsList[intIndex].VarName));
						THIS^.M_LogMessage(CONCAT(aExpectedOutputParamsList[intIndex].VarName,CONCAT(' Int Parameter is ', DINT_TO_STRING(intValue))));
						_inst_strlocal := DINT_TO_STRING(intValue);
						aoutputParam[intIndex].strValue := _inst_strlocal;
					ELSIF aExpectedOutputParamsList[intIndex].DataType = E_DataType.DT_UINT THEN
						uintValue := _inst_fbParams.M_ParseUint(_inst_fbParams.M_GetStructMember(_pStructPointerAbs,aExpectedOutputParamsList[intIndex].VarName));
						THIS^.M_LogMessage(CONCAT(aExpectedOutputParamsList[intIndex].VarName,CONCAT(' Uint Parameter is ', UDINT_TO_STRING(uintValue))));
						_inst_strlocal := UDINT_TO_STRING(uintValue);
						aoutputParam[intIndex].strValue := _inst_strlocal;
					ELSIF aExpectedOutputParamsList[intIndex].DataType = E_DataType.DT_ULINT THEN
						ulintValue := _inst_fbParams.M_ParseUint64(_inst_fbParams.M_GetStructMember(_pStructPointerAbs,aExpectedOutputParamsList[intIndex].VarName));
						THIS^.M_LogMessage(CONCAT(aExpectedOutputParamsList[intIndex].VarName,CONCAT(' ULINT Parameter is ', ULINT_TO_STRING(ulintValue))));
						_inst_strlocal := ULINT_TO_STRING(ulintValue);
						aoutputParam[intIndex].strValue := _inst_strlocal;
					ELSIF aExpectedOutputParamsList[intIndex].DataType = E_DataType.DT_DOUBLE THEN
						floatResponse := _inst_fbParams.M_ParseDouble(_inst_fbParams.M_GetStructMember(_pStructPointerAbs,aExpectedOutputParamsList[intIndex].VarName));
						THIS^.M_LogMessage(CONCAT(aExpectedOutputParamsList[intIndex].VarName,CONCAT(' float Parameter is ', LREAL_TO_STRING(floatResponse)))); 
						aoutputParam[intIndex].strValue := LREAL_TO_STRING(floatResponse);
					ELSIF aExpectedOutputParamsList[intIndex].DataType = E_DataType.DT_BOOL THEN
						boolresponse := _inst_fbParams.M_ParseBool(_inst_fbParams.M_GetStructMember(_pStructPointerAbs,aExpectedOutputParamsList[intIndex].VarName));
						THIS^.M_LogMessage(CONCAT(aExpectedOutputParamsList[intIndex].VarName, CONCAT(' Bool Response is ',BOOL_TO_STRING(boolresponse))));
						aoutputParam[intIndex].strValue := BOOL_TO_STRING(boolresponse);						
					ELSE
						aoutputParam[intIndex].strValue :=_inst_fbParams.M_ParseString(_inst_fbParams.M_GetStructMember(_pStructPointerAbs,aExpectedOutputParamsList[intIndex].VarName));
						THIS^.M_LogMessage(CONCAT(aExpectedOutputParamsList[intIndex].VarName,CONCAT(' String Parameter is ', aoutputParam[intIndex].strValue)));	
					END_IF
				END_IF
			END_FOR	
		// Set error if command failed
		ELSE
			THIS^.M_SetError(_udintERROR_ID, _strERROR_MSG);
		END_IF
		// Go back to start
		_inst_intStep := 0;
END_CASE
M_RunCommand := _bResult;
intMRunCommandStep := _inst_intStep;
END_METHOD

METHOD M_RunImpMethods : BOOL
VAR_INPUT
    
END_VAR

VAR CONSTANT
	_strCOMMAND_NAME : T_MaxString	:= 'RunImpMethods'; // Name of the API method
	_timeCOMMAND_TIMEOUT : TIME		:= T#5S; // Max time to receive API response
	_strSTART_MSG : T_MaxString		:= 'Runs Imp Methods on DeviceComm Class'; // Prints when method starts
	_strEND_MSG : T_MaxString		:= 'RunImpMethod succesfull'; // Prints when method finishes
	_udintERROR_ID : UDINT			:= E_COHAP_Error.FailedToRunImpMethods; // Error ID to set if command fails
	_strERROR_MSG : T_MaxString		:= 'RunImpMethods Failed!'; // Error message to set if command fails
END_VAR
VAR_INST
	_inst_arrParams: T_ApiParameterList; // Parameters array
	_inst_arrOutputs: T_ApiParameterList; // Outputs array
	_inst_strRet: T_ApiParamValue; // Return string from the router
	_inst_intStep: INT; // Current method step
	_inst_fbParams: FB_ApiParamBuilder; // Parameter builder FB
END_VAR
VAR
	_bComplete: BOOL; // True if the routing finishes
	_intRet: INT; // Return string converted to an integer
	_bResult : BOOL; // Output of the method
END_VAR
_inst_intStep:=intMRunImpMethodsStep;
bRunImpMethodsBusy:=TRUE;

_bResult := FALSE;
CASE _inst_intStep OF
	0: // Wait for no error and router not busy
		IF NOT THIS^.P_bError AND NOT bRouterBusy THEN
			bRouterBusy := TRUE;
			_inst_intStep := _inst_intStep + 10;
		END_IF
		
	10: // Initialize parameters
		THIS^.M_LogMessage(_strSTART_MSG);
		_inst_fbParams.M_ClearParameters();
		// ADD ANY PARAMETERS HERE
//		_inst_fbParams.M_AddParameter('devID', strDevName);
		
		_inst_fbParams.M_OutputToParameterList(_inst_arrParams);
		_inst_intStep := _inst_intStep + 10;
		
	20: // Route the command
		_bComplete := M_RouterHelper(
			_in_strMethodName := _strCOMMAND_NAME, 
			_in_timeTimeout := _timeCOMMAND_TIMEOUT,
			_inout_arrParams := _inst_arrParams,
			_inout_arrOutputs := _inst_arrOutputs,
			_out_strReturnValue=>_inst_strRet);
		
		// If route completed, move to next step
		IF _bComplete THEN
			_inst_intStep := _inst_intStep + 10;
			bRouterBusy := FALSE;
		ELSIF THIS^.P_bError THEN
			_inst_intStep := 0;
			bRouterBusy := FALSE;
		END_IF
		
	30: // Parse results
		_intRet := STRING_TO_INT(_inst_strRet);
		IF _intRet > 0 THEN
			_bResult := TRUE;
			THIS^.M_LogMessage(_strEND_MSG);
			// DO ANY PARSING HERE
			_inst_fbParams.M_LoadFromParameterList(_inst_arrOutputs);
		
		// Set error if command failed
	
		ELSE
			THIS^.M_SetError(_udintERROR_ID, _strERROR_MSG);
		END_IF
		
		// Go back to start
		_inst_intStep := 0;
END_CASE
M_RunImpMethods := _bResult;
intMRunImpMethodsStep :=_inst_intStep;
END_METHOD

END_FUNCTION_BLOCK

// Project Information/F_GetCompany
// This function has been automatically generated from the project information.
{attribute 'signature_flag' := '1073741824'}
{attribute 'TcGenerated'}
{attribute 'no-analysis'}
FUNCTION F_GetCompany : WSTRING
VAR_INPUT
	
END_VAR

F_GetCompany := "Sensata Technologies";

END_FUNCTION

// Project Information/F_GetTitle
// This function has been automatically generated from the project information.
{attribute 'signature_flag' := '1073741824'}
{attribute 'TcGenerated'}
{attribute 'no-analysis'}
FUNCTION F_GetTitle : WSTRING
VAR_INPUT
	
END_VAR

F_GetTitle := "Sensata_Device_Comm";

END_FUNCTION

// Project Information/F_GetVersion
// This function has been automatically generated from the project information.
{attribute 'signature_flag' := '1073741824'}
{attribute 'TcGenerated'}
{attribute 'no-analysis'}
FUNCTION F_GetVersion : ST_LibVersion
VAR_INPUT
	
END_VAR

F_GetVersion.iMajor := 0;
F_GetVersion.iMinor := 0;
F_GetVersion.iBuild := 1;
F_GetVersion.iRevision := 0;
F_GetVersion.sVersion := '0.0.1';
F_GetVersion.nFlags := 0;

END_FUNCTION
